{attribute 'GeneratedUsingTerminal: EK1122-0000-0018'}
{attribute addProperty BoxType "EK1122-0000-0018"}
{attribute addProperty Id "Beckhoff_EL3xxx_0030sub_EK1100EK1100_AB5A94672"}
{attribute addProperty CRC "3152050556"}
{attribute addProperty Size "2"}
TYPE Beckhoff_EL3xxx_0030EK1122_BBE0797C EXTENDS EK1122_AB5A9467 :
STRUCT
	{attribute addProperty Name "Beckhoff_EL3xxx_0030sub_EK1100"}
	Beckhoff_EL3xxx_0030sub_EK1100 : EK1100_AB5A9467;
END_STRUCT
END_TYPE

(* stored: Version 1.2.0.0, ProductVersion 3.1.4024.9
   DUT Beckhoff_EL3xxx_0030EK1122_BBE0797C: Id {dba9b122-d370-44ae-88c7-95fa59754bcd} *)
